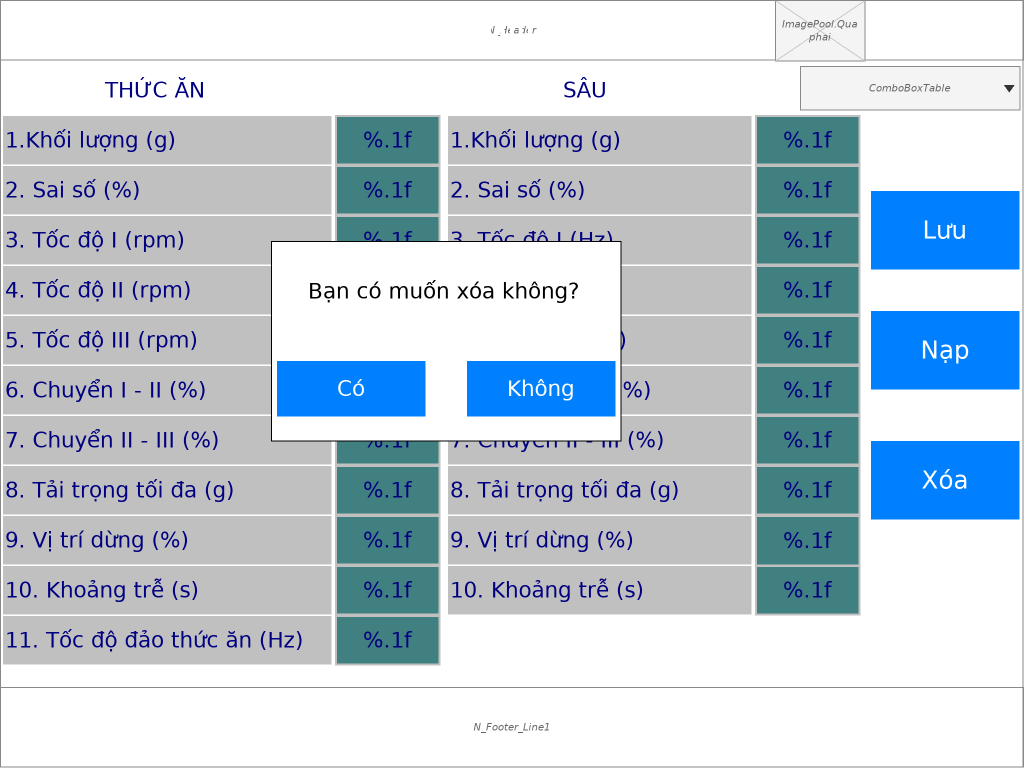
VISUALIZATION N_Recipe_Line1  // 1024x768
    Frame (0,687 1024x80)
        shows N_Footer_Line1()
    Frame (0,0 1024x60)
        shows N_Header()
    Textfield (353,5 400x50), "MÀN HÌNH LƯU THÔNG SỐ LINE 1"
    Textfield (80,75 150x30), "THỨC ĂN"
    Textfield (545,75 80x30), "SÂU"
    Rectangle (870,190 150x80), "Lưu"
        tap GVL_OF_VU.bRecSave[1]
        OnDialogClosed: execute { bSave1 := true; }
        OnMouseClick: write PRG_MainRecipe1.NameSave via VisuDialogs.Keypad
    Rectangle (870,440 150x80), "Xóa"
        tap GVL_OF_VU.bRecDelete[1]
        OnMouseDown: execute { GVL_OF_VU.bDeleteRecipe1 := TRUE; }
    Rectangle (870,310 150x80), "Nạp"
        tap GVL_OF_VU.bRecLoad[1]
        OnMouseDown: execute { bLoad1 := true; }
    ComboBoxTable (800,66 220x44), variable: PRG_MainRecipe1.RecipeNameIdx, data array: PRG_MainRecipe1.RecipeList
        p3854506369: PRG_MainRecipe1.RecipeList[INDEX]
    Rectangle (447,115 305x50), "1.Khối lượng (g)"
    Rectangle (447,165 305x50), "2. Sai số (%)"
    Rectangle (447,215 305x50), "3. Tốc độ I (Hz)"
    Rectangle (447,265 305x50), "4. Tốc độ II (Hz)"
    Rectangle (447,365 305x50), "6. Chuyển I - II (%)"
    Rectangle (447,465 305x50), "8. Tải trọng tối đa (g)"
    Rectangle (447,315 305x50), "5. Tốc độ III (Hz)"
    Rectangle (447,415 305x50), "7. Chuyển II - III (%)"
    Rectangle (447,565 305x50), "10. Khoảng trễ (s)"
    Rectangle (447,515 305x50), "9. Vị trí dừng (%)"
    Rectangle (2,115 330x50), "1.Khối lượng (g)"
    Rectangle (2,165 330x50), "2. Sai số (%)"
    Rectangle (2,215 330x50), "3. Tốc độ I (rpm)"
    Rectangle (2,265 330x50), "4. Tốc độ II (rpm)"
    Rectangle (2,365 330x50), "6. Chuyển I - II (%)"
    Rectangle (2,465 330x50), "8. Tải trọng tối đa (g)"
    Rectangle (2,315 330x50), "5. Tốc độ III (rpm)"
    Rectangle (2,415 330x50), "7. Chuyển II - III (%)"
    Rectangle (2,565 330x50), "10. Khoảng trễ (s)"
    Rectangle (2,515 330x50), "9. Vị trí dừng (%)"
    Rectangle (2,615 330x50), "11. Tốc độ đảo thức ăn (Hz)"
    Image (775,0 90x61), image: ImagePool.Qua phai
        OnMouseClick: change screen: N_Recipe_Line2
    Textfield (335,115 105x50), "%.1f", text variable: PR_Line01.fDerisedWeight_Food
    Textfield (335,165 105x50), "%.1f", text variable: PR_Line01.fDelta_Food
    Textfield (335,215 105x50), "%.1f", text variable: PR_Line01.fFast_Speed
    Textfield (335,265 105x50), "%.1f", text variable: PR_Line01.fSlow_Speed_1
    Textfield (335,315 105x50), "%.1f", text variable: PR_Line01.fSlow_Speed_2
    Textfield (335,365 105x50), "%.1f", text variable: PR_Line01.fChangeMode_Food_1
    Textfield (335,415 105x50), "%.1f", text variable: PR_Line01.fChangeMode_Food_2
    Textfield (335,465 105x50), "%.1f", text variable: PR_Line01.fMaxWeight_Food
    Textfield (335,515 105x50), "%.1f", text variable: PR_Line01.fPerStop_Food
    Textfield (335,565 105x50), "%.1f", text variable: PR_Line01.fTimer_Check_Food
    Textfield (335,615 105x50), "%.1f", text variable: PR_Line01.fSpeed_motor_mixer
    Textfield (755,115 105x50), "%.1f", text variable: PR_Line01.fDerisedWeight_Worm
    Textfield (755,165 105x50), "%.1f", text variable: PR_Line01.fDelta_Worm
    Textfield (755,215 105x50), "%.1f", text variable: PR_Line01.fFast_Speed_vibrating_funnel
    Textfield (755,265 105x50), "%.1f", text variable: PR_Line01.fSlow_Speed_vibrating_funnel_1
    Textfield (755,315 105x50), "%.1f", text variable: PR_Line01.fSlow_Speed_vibrating_funnel_2
    Textfield (755,365 105x50), "%.1f", text variable: PR_Line01.fChangeMode_Worm_1
    Textfield (755,415 105x50), "%.1f", text variable: PR_Line01.fChangeMode_Worm_2
    Textfield (755,465 105x50), "%.1f", text variable: PR_Line01.fMaxWeight_Worm
    Textfield (755,515 105x51), "%.1f", text variable: PR_Line01.fPerStop_Worm
    Textfield (755,565 105x50), "%.1f", text variable: PR_Line01.fTimer_Check_Worm
    GroupBox (271,241 350x200), invisible if: not GVL_OF_VU.bDeleteRecipe1, input disabled if: not GVL_OF_VU.bDeleteRecipe1
        Rectangle (0,0 350x200)
        Rectangle (5,119 150x57), "Có"
            OnMouseDown: execute { bDelete1 := true; }
            OnMouseUp: execute { GVL_OF_VU.bDeleteRecipe1 := FALSE; }
        Label (4,29 338x42), "Bạn có muốn xóa không?"
        Rectangle (195,119 150x57), "Không"
            OnMouseDown: execute { GVL_OF_VU.bDeleteRecipe1 := FALSE; }
END_VISUALIZATION

(* stored: Version 1.1.0.1, ProductVersion 3.1.4024.12
   Visu N_Recipe_Line1: Id {4202c50c-2d16-4b9a-9d32-eeda31856d2e} *)
